// TIA Portal V16 export
// export: Created 2023-03-29T11:03:30.1712239Z, ExportSetting WithDefaults, DisplayName Totally Integrated Automation Portal, DisplayVersion V16 Update 6, DisplayName TIA Portal Version Control Interface, DisplayVersion V16 Update 2, DisplayName TIA Portal Openness, DisplayVersion V16 Update 6, DisplayName STEP 7 Professional, DisplayVersion V16 Update 6, DisplayName STEP 7 Safety, DisplayVersion V16, DisplayName WinCC Advanced, DisplayVersion V16 Update 6
DATA_BLOCK "VLV02_DB_Z8"   // DB20
AUTHOR : RTecmer
VERSION : 0.2
// stored: AutoNumber true, DBAccessibleFromOPCUA true, InstanceOfName VLV02, InstanceOfType FB
"VLV02"
   // VAR_INPUT
   //    SVMC : Bool;
   //    SVMO { ExternalVisible := 'False'} : Bool;
   //    CLSD : Bool;
   //    OPND : Bool;
   //    REMT : Bool;
   //    KT1 : Time;
   // END_VAR
   // VAR_IN_OUT
   //    CLSE { ExternalAccessible := 'False'; ExternalVisible := 'False'; ExternalWritable := 'False'} : Bool;
   //    OPEN { ExternalAccessible := 'False'; ExternalVisible := 'False'; ExternalWritable := 'False'} : Bool;
   //    WIZ : Byte;
   //    STAT : Byte;
   //    TMR1 : TON_TIME;
   // END_VAR
BEGIN
END_DATA_BLOCK
